(* PLC project Singleton1, Beckhoff Automation GmbH TwinCAT PLC Control 3.5.13.21 *)
(* stored: creationDateTime 2023-12-23T12:40:08.3527674, modificationDateTime 2023-12-23T12:40:08.3605762 *)

{attribute 'qualified_only'}
{attribute 'strict'}
TYPE E_Color :
(
	NoColor := 0,
	Blue,
	Green,
	Yellow
	
);
END_TYPE

INTERFACE Proxy_Interface
///Illustrative method of the pattern
METHOD Set_Background
VAR_INPUT
	///HEX value to be set as background color
	newBackground: DWORD;
END_VAR
END_METHOD
END_INTERFACE

PROGRAM PLC_PRG
VAR
	///Blue, highly opaque
	dwBlue: DWORD := 16#FF0000FF;
	///Green, highly opaque
	dwGreen: DWORD := 16#FF00FF00;
	///Yellow, highly opaque
	dwYellow: DWORD := 16#FFFFFF00;
	///Creates 3 instances of the ProxyToSingleton class
	instance1: ProxyToSingleton;
	instance2: ProxyToSingleton;
	instance3: ProxyToSingleton;
	
	eInstance1 : E_Color;
	eInstance2 : E_Color;
	eInstance3 : E_Color;
	
END_VAR

                  //*************************************************************************************************************************************************************
//The PLC_PRG handles the instanciation of the possible background colours and the ProxyToSingleton instances in order to be used by the Visualization element.
//The viasualization element (The client) handles the request for background change on the RealSingleton object through the ProxyToSinlgeton instances.
//These request are first processed by the ProxyToSingleton object and then passed to the one and only RealSingleton instance.
//The default background colour of the RealSingleton object is 'Blue' 
//*************************************************************************************************************************************************************
// spanish
//PLC_PRG maneja la instanciación de los posibles colores de fondo y las instancias de ProxyToSingleton para ser utilizados por el elemento de visualización.
//El elemento de visualización (el cliente) maneja la solicitud de cambio de fondo en el objeto RealSingleton a través de las instancias de ProxyToSinlgeton.
//Estas solicitudes son procesadas primero por el objeto ProxyToSingleton y luego pasadas a la única instancia de RealSingleton.
//El color de fondo predeterminado del objeto RealSingleton es 'Azul'
//*************************************************************************************************************************************************************

CASE eInstance1 OF
	E_Color.Blue:
		instance1.Set_Background(dwBlue);
		eInstance1:=E_Color.NoColor;
	E_Color.Green:
		instance1.Set_Background(dwGreen);
		eInstance1:=E_Color.NoColor;
	E_Color.Yellow:
		instance1.Set_Background(dwYellow);
		eInstance1:=E_Color.NoColor;
END_CASE

CASE eInstance2 OF
	E_Color.Blue:
		instance2.Set_Background(dwBlue);
		eInstance2:=E_Color.NoColor;	
	E_Color.Green:
		instance2.Set_Background(dwGreen);
		eInstance2:=E_Color.NoColor;	
	E_Color.Yellow:
		instance2.Set_Background(dwYellow);
		eInstance2:=E_Color.NoColor;	
END_CASE

CASE eInstance3 OF
	E_Color.Blue:
		instance3.Set_Background(dwBlue);
		eInstance3:=E_Color.NoColor;	
	E_Color.Green:
		instance3.Set_Background(dwGreen);
		eInstance3:=E_Color.NoColor;	
	E_Color.Yellow:
		instance3.Set_Background(dwYellow);
		eInstance3:=E_Color.NoColor;	
END_CASE
                
END_PROGRAM

/// ****************************************************************************************************************************************
/// This class is called ProxyToSingleton because it works as a Proxy of the Singleton class. It handles the creation and instanciation of the 
/// RealSingleton class. Something like the proper static method GetInstance(); in any singleton pattern.
/// So the ProxyToSingleton class has a static Singleton object as a field and whenever we instanciate a 
/// ProxyToSingleton object we will have the RealSingleton object as its static field .realSingleton^
/// ****************************************************************************************************************************************
/// Spanish
/// Esta clase se llama ProxyToSingleton porque funciona como Proxy de la clase Singleton. Se encarga de la creación e instanciación de la
/// Clase RealSingleton. Algo así como el método estático adecuado GetInstance(); en cualquier patrón singleton.
/// Entonces la clase ProxyToSingleton tiene un objeto Singleton estático como campo y cada vez que instanciamos un
/// Objeto ProxyToSingleton tendremos el objeto RealSingleton como su campo estático .realSingleton^
/// ****************************************************************************************************************************************
{attribute 'enable_dynamic_creation' := ''}
FUNCTION_BLOCK ProxyToSingleton IMPLEMENTS Proxy_Interface
VAR_STAT
	///Boolean value to check if there is already a Singleton instance
	//****************************************************************
	///Valor booleano para comprobar si ya existe una instancia Singleton
	bFirstInstance: BOOL := FALSE;
	///Pointer to the first and only instance of the Singleton class
	//***************************************************************
	///Puntero a la primera y única instancia de la clase Singleton
	realSingleton: POINTER TO RealSingleton;
END_VAR

                  
                

METHOD fb_init
VAR_INPUT
	/// TRUE: the Retain-variables are initialized (reset warm / reset cold)
	bInitRetains: BOOL;
	/// TRUE  the instance will be copied to the copy-code afterward (online change)
	bInCopyCode: BOOL;
END_VAR
                        //THIS FUNCTION WORKS AS THE CONSTRUCTOR OF THE ProxyToSingleton CLASS
// It handles the creation of the only RealSingleton object. It uses the concept of lazy instanciation.

//If the static property .bFirstInstance is TRUE
//*********************************************************************************************************
//ESTA FUNCIÓN FUNCIONA COMO CONSTRUCTOR DE LA CLASE ProxyToSingleton
// Maneja la creación del único objeto RealSingleton. Utiliza el concepto de instanciación diferida.

//Si la propiedad estática .bFirstInstance es VERDADERA
IF THIS^.bFirstInstance = TRUE
	
THEN
		// There is already a Singleton object.
		// So we don't have to do anything, this new ProxyToSingleton object will already have the address of the 
		// RealSingleton object in its pointer .realSingleton
		//*********************************************************************************************************
		// Ya existe un objeto Singleton.
		// Así que no tenemos que hacer nada, este nuevo objeto ProxyToSingleton ya tendrá la dirección del
		// objeto RealSingleton en su puntero .realSingleton
	
	ELSE	
		//If the static property .bFirstInstance is FALSE
		//*************************************************
		//Si la propiedad estática .bFirstInstance es FALSA
	
		// There is not a Singleton object so the ProxyToSingleton object calling the constructor 
		// should create the RealSingleton object in its pointer field .realSingleton 
		// Then we change the status of the static variable bFirstInstance to TRUE and avoid overwriting the realSingleton address.
		// If the Singleton object is destroyed, .bFirstInstance should be set to FALSE again.
		//************************************************************************************************************************
		// No hay un objeto Singleton, por lo que el objeto ProxyToSingleton llama al constructor
		// debería crear el objeto RealSingleton en su campo de puntero .realSingleton
		// Luego cambiamos el estado de la variable estática bFirstInstance a TRUE y evitamos sobrescribir la dirección realSingleton.
		// Si el objeto Singleton se destruye, .bFirstInstance debe establecerse en FALSO nuevamente.
		THIS^.bFirstInstance := TRUE;
		
		// Reference the value of the first RealSingleton instance to the FakeSingleton object to save 
		// the address of the real Singleton instance.
		// *****************************************************************************************
		// Referencia el valor de la primera instancia de RealSingleton al objeto FakeSingleton para guardar
		// la dirección de la instancia Singleton real.
		THIS^.realSingleton := __NEW(RealSingleton);
END_IF
                      
END_METHOD

///Illustrative method of the pattern
METHOD Set_Background
VAR_INPUT
	///HEX value to be set as background color
	newBackground: DWORD;
END_VAR
                        //The ProxyToSingleton object handles the request and send the appropiate reques to the one and only RealSingleton instance
//**************************************************************************************************************************
//El objeto ProxyToSingleton maneja la solicitud y envía las solicitudes apropiadas a la única instancia de RealSingleton
THIS^.realSingleton^.Set_Background(newBackground);

                      
END_METHOD
END_FUNCTION_BLOCK

///*****************************************************************************************************************
/// This class is called RealSingleton because it works as singleton.  
/// As long as we only instanciate ProxyToSingleton objects, this class will work as a Singleton class should work.
/// The global access point to this class is the field .realSingleton^ in every ProxyToSingleton object.
///*****************************************************************************************************************
/// Esta clase se llama RealSingleton porque funciona como singleton.
/// Siempre que solo instanciamos objetos ProxyToSingleton, esta clase funcionará como debería funcionar una clase Singleton.
/// El punto de acceso global a esta clase es el campo .realSingleton^ en cada objeto ProxyToSingleton.
///*****************************************************************************************************************
{attribute 'enable_dynamic_creation' := ''}
FUNCTION_BLOCK RealSingleton IMPLEMENTS Proxy_Interface
VAR
	///Illustrative field of the pattern to store the HEX value for the background colour
	///************************************************************************************
	///Campo ilustrativo del patrón para almacenar el valor HEX para el color de fondo	
	backgroundColour: DWORD;
END_VAR

                  
                

METHOD fb_init
VAR_INPUT
	/// TRUE: the Retain-variables are initialized (reset warm / reset cold)
	bInitRetains: BOOL;
	/// TRUE  the instance will be copied to the copy-code afterward (online change)
	bInCopyCode: BOOL;
END_VAR
                        //The default valur for the background is set
//*********************************************
//Se establece el valor predeterminado para el fondo
THIS^.Set_Background(PLC_PRG.dwBlue);

                      
END_METHOD

///Illustrative method of the pattern
METHOD Set_Background
VAR_INPUT
	///HEX value to be set as background color
	newBackground: DWORD;
END_VAR
                        //Writes the backgroundColour field to the passed newBackground value
//********************************************************************
//Escribe el campo backgroundColor en el valor newBackground pasado
THIS^.backgroundColour := newBackground;
                      
END_METHOD
END_FUNCTION_BLOCK

PROGRAM MAIN
VAR
END_VAR

                  PLC_PRG();
                
END_PROGRAM

CONFIGURATION Application
  RESOURCE Singleton1 ON PLC
    TASK PlcTask(INTERVAL := T#0ms, PRIORITY := 20);
    PROGRAM MAIN WITH PlcTask : MAIN;
  END_RESOURCE
END_CONFIGURATION
